// TIA Portal V20 export
DATA_BLOCK "Simulation_DB"   // DB184
// stored: InstanceOfName Unit1.Em3.Simulation, InstanceOfType FB, Namespace Unit1.Em3
"Unit1.Em3.Simulation"
   // VAR_INPUT
   //    simulation { ExternalAccessible := 'False'; ExternalVisible := 'False'; ExternalWritable := 'False'} : Bool;
   // END_VAR
   // VAR
   //    instActuator { ExternalAccessible := 'False'; ExternalVisible := 'False'; ExternalWritable := 'False'} : Array[0..19] of "Simulation_Actuator";
   //    statDigitalSignal { ExternalAccessible := 'False'; ExternalVisible := 'False'; ExternalWritable := 'False'} : Array[0..9] of Bool;
   // END_VAR
BEGIN
END_DATA_BLOCK
